(* Logix 5000 project; controller Week_4_PLC_1_AND_Condition Emulate 5570 rev 30.12; software revision 30.01 *)

TASK MainTask (continuous, watchdog 500 ms) : MainProgram

MODULES
   Local : Emulate 5570 (ICP 2, rev 30.12)
END_MODULES

PROGRAM MainProgram   (* main routine MainRoutine *)
VAR
   Counter : COUNTER := (PRE := 10);
   Output1 : BOOL;
   PB1 : BOOL;
END_VAR

ROUTINE MainRoutine   (* ladder *)
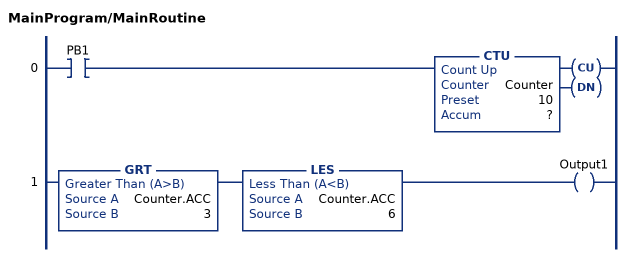
   0: XIC(PB1)CTU(Counter,?,?);
   1: GRT(Counter.ACC,3)LES(Counter.ACC,6)OTE(Output1);
END_ROUTINE
END_PROGRAM
